FUNCTION Convert_LWORD_TO_BYTE : Hresult
VAR_INPUT
	in : LWORD;
	out : REFERENCE TO BYTE;
END_VAR
VAR
	converted : BYTE;
END_VAR
VAR CONSTANT
	INCOMPATIBLE : HRESULT := 16#9811070E;
END_VAR

converted := LWORD_TO_BYTE(in);

IF (BYTE_TO_LWORD(converted) <> in) THEN
	Convert_LWORD_TO_BYTE := INCOMPATIBLE;
	RETURN;
END_IF

out := converted;

END_FUNCTION

(* stored: Version 1.1.0.1, ProductVersion 3.1.4024.12
   POU Convert_LWORD_TO_BYTE: Id {73d2cd9b-9f23-4ee2-b369-5b97de2acc42}, SpecialFunc None *)
